TYPE ST_KPI_InspectionEfficency :
STRUCT
	ProcessedTotal			: UDINT;
	ProcessedSuccessful		: UDINT;
	ProcessedRejected		: UDINT;
	ProcessedEfficiency		: LREAL;
END_STRUCT
END_TYPE

(* stored: Version 1.1.0.1
   DUT ST_KPI_InspectionEfficency: Id {c1c58aeb-35be-4790-a746-7873a1528bfe} *)
